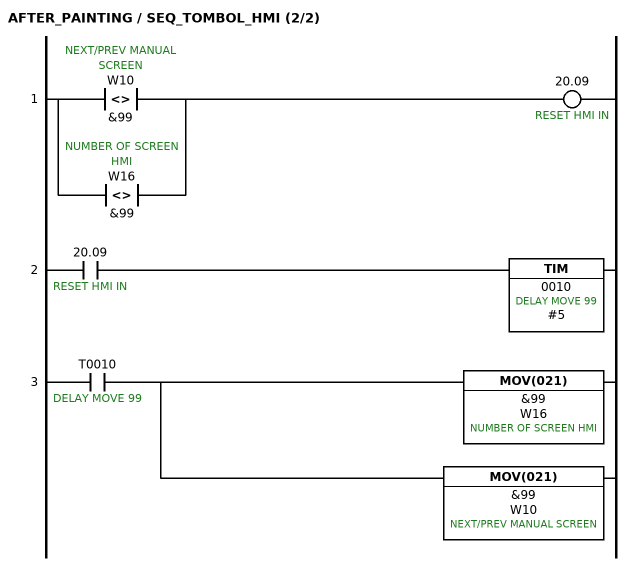
; [picture p48: AFTER_PAINTING / SEQ_TOMBOL_HMI, rungs 1-3]
; rung 1
LD<>(305) W10 &99  ; NEXT/PREV MANUAL SCREEN
OR<>(305) W16 &99  ; NUMBER OF SCREEN HMI
OUT 20.09  ; RESET HMI IN
; rung 2
LD 20.09  ; RESET HMI IN
TIM 0010 #5  ; DELAY MOVE 99
; rung 3
LD T0010  ; DELAY MOVE 99
MOV(021) &99 W16  ; NUMBER OF SCREEN HMI
MOV(021) &99 W10  ; NEXT/PREV MANUAL SCREEN

### Section AUTI

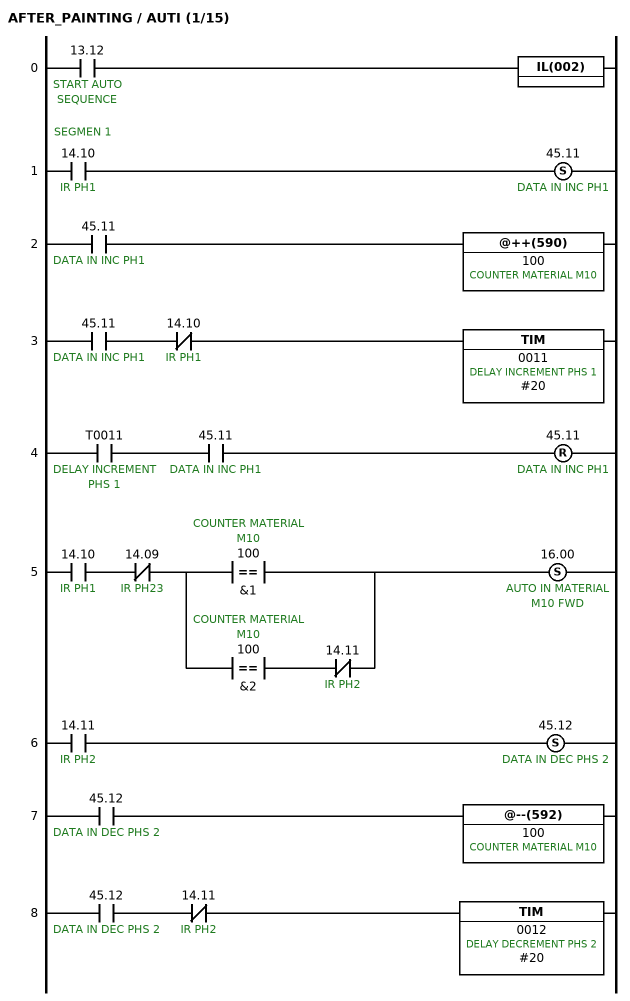
; rung 0
LD 13.12  ; START AUTO SEQUENCE
IL(002)
; rung 1: SEGMEN 1
LD 14.10  ; IR PH1
SET 45.11  ; DATA IN INC PH1
; rung 2
LD 45.11  ; DATA IN INC PH1
@++(590) 100  ; COUNTER MATERIAL M10
; rung 3
LD 45.11  ; DATA IN INC PH1
ANDNOT 14.10  ; IR PH1
TIM 0011 #20  ; DELAY INCREMENT PHS 1
; rung 4
LD T0011  ; DELAY INCREMENT PHS 1
AND 45.11  ; DATA IN INC PH1
RSET 45.11  ; DATA IN INC PH1
; rung 5
LD 14.10  ; IR PH1
ANDNOT 14.09  ; IR PH23
LD=(300) 100 &1  ; COUNTER MATERIAL M10
LD=(300) 100 &2  ; COUNTER MATERIAL M10
ANDNOT 14.11  ; IR PH2
ORLD
ANDLD
SET 16.00  ; AUTO IN MATERIAL M10 FWD
; rung 6
LD 14.11  ; IR PH2
SET 45.12  ; DATA IN DEC PHS 2
; rung 7
LD 45.12  ; DATA IN DEC PHS 2
@--(592) 100  ; COUNTER MATERIAL M10
; rung 8
LD 45.12  ; DATA IN DEC PHS 2
ANDNOT 14.11  ; IR PH2
TIM 0012 #20  ; DELAY DECREMENT PHS 2

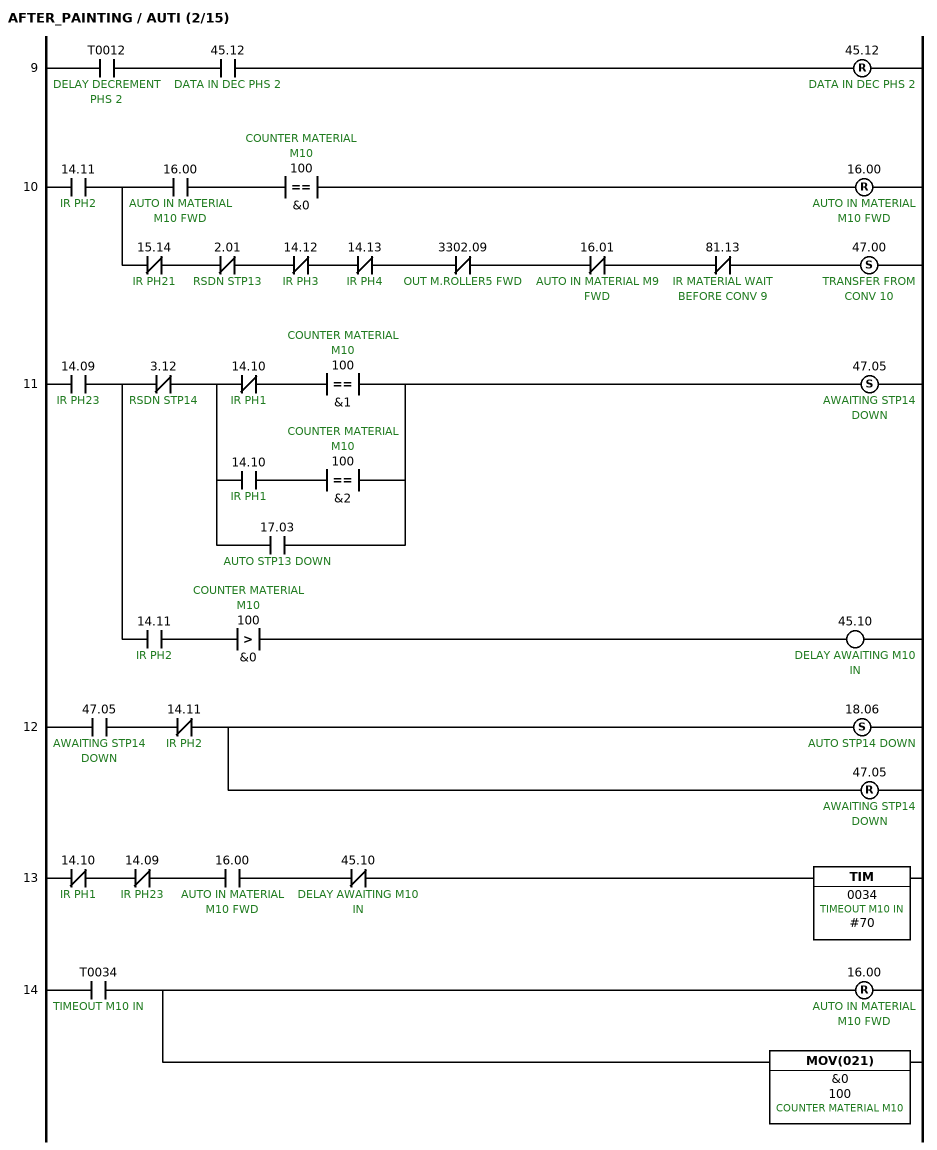
; rung 9
LD T0012  ; DELAY DECREMENT PHS 2
AND 45.12  ; DATA IN DEC PHS 2
RSET 45.12  ; DATA IN DEC PHS 2
; rung 10
LD 14.11  ; IR PH2
OUT TR0
AND 16.00  ; AUTO IN MATERIAL M10 FWD
AND=(300) 100 &0  ; COUNTER MATERIAL M10
RSET 16.00  ; AUTO IN MATERIAL M10 FWD
LD TR0
ANDNOT 15.14  ; IR PH21
ANDNOT 2.01  ; RSDN STP13
ANDNOT 14.12  ; IR PH3
ANDNOT 14.13  ; IR PH4
ANDNOT 3302.09  ; OUT M.ROLLER5 FWD
ANDNOT 16.01  ; AUTO IN MATERIAL M9 FWD
ANDNOT 81.13  ; IR MATERIAL WAIT BEFORE CONV 9
SET 47.00  ; TRANSFER FROM CONV 10
; rung 11
LD 14.09  ; IR PH23
OUT TR0
ANDNOT 3.12  ; RSDN STP14
LDNOT 14.10  ; IR PH1
AND=(300) 100 &1  ; COUNTER MATERIAL M10
LD 14.10  ; IR PH1
AND=(300) 100 &2  ; COUNTER MATERIAL M10
ORLD
OR 17.03  ; AUTO STP13 DOWN
ANDLD
SET 47.05  ; AWAITING STP14 DOWN
LD TR0
AND 14.11  ; IR PH2
AND>(320) 100 &0  ; COUNTER MATERIAL M10
OUT 45.10  ; DELAY AWAITING M10 IN
; rung 12
LD 47.05  ; AWAITING STP14 DOWN
ANDNOT 14.11  ; IR PH2
SET 18.06  ; AUTO STP14 DOWN
RSET 47.05  ; AWAITING STP14 DOWN
; rung 13
LDNOT 14.10  ; IR PH1
ANDNOT 14.09  ; IR PH23
AND 16.00  ; AUTO IN MATERIAL M10 FWD
ANDNOT 45.10  ; DELAY AWAITING M10 IN
TIM 0034 #70  ; TIMEOUT M10 IN
; rung 14
LD T0034  ; TIMEOUT M10 IN
RSET 16.00  ; AUTO IN MATERIAL M10 FWD
MOV(021) &0 100  ; COUNTER MATERIAL M10

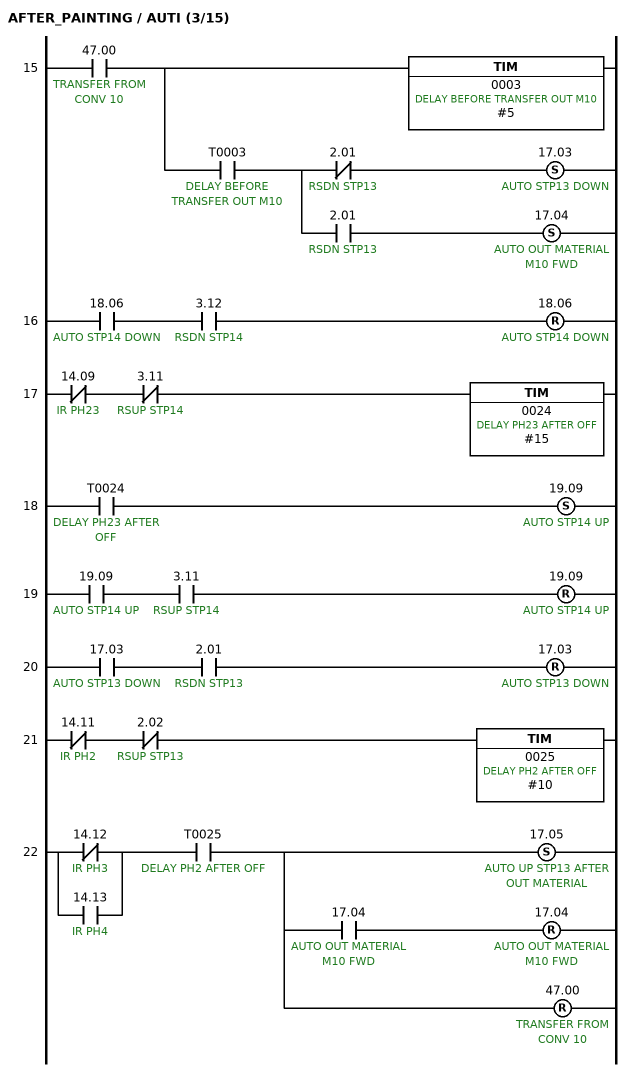
; rung 15
LD 47.00  ; TRANSFER FROM CONV 10
TIM 0003 #5  ; DELAY BEFORE TRANSFER OUT M10
AND T0003  ; DELAY BEFORE TRANSFER OUT M10
OUT TR0
ANDNOT 2.01  ; RSDN STP13
SET 17.03  ; AUTO STP13 DOWN
LD TR0
AND 2.01  ; RSDN STP13
SET 17.04  ; AUTO OUT MATERIAL M10 FWD
; rung 16
LD 18.06  ; AUTO STP14 DOWN
AND 3.12  ; RSDN STP14
RSET 18.06  ; AUTO STP14 DOWN
; rung 17
LDNOT 14.09  ; IR PH23
ANDNOT 3.11  ; RSUP STP14
TIM 0024 #15  ; DELAY PH23 AFTER OFF
; rung 18
LD T0024  ; DELAY PH23 AFTER OFF
SET 19.09  ; AUTO STP14 UP
; rung 19
LD 19.09  ; AUTO STP14 UP
AND 3.11  ; RSUP STP14
RSET 19.09  ; AUTO STP14 UP
; rung 20
LD 17.03  ; AUTO STP13 DOWN
AND 2.01  ; RSDN STP13
RSET 17.03  ; AUTO STP13 DOWN
; rung 21
LDNOT 14.11  ; IR PH2
ANDNOT 2.02  ; RSUP STP13
TIM 0025 #10  ; DELAY PH2 AFTER OFF
; rung 22
LDNOT 14.12  ; IR PH3
OR 14.13  ; IR PH4
AND T0025  ; DELAY PH2 AFTER OFF
OUT TR0
SET 17.05  ; AUTO UP STP13 AFTER OUT MATERIAL
AND 17.04  ; AUTO OUT MATERIAL M10 FWD
RSET 17.04  ; AUTO OUT MATERIAL M10 FWD
LD TR0
RSET 47.00  ; TRANSFER FROM CONV 10

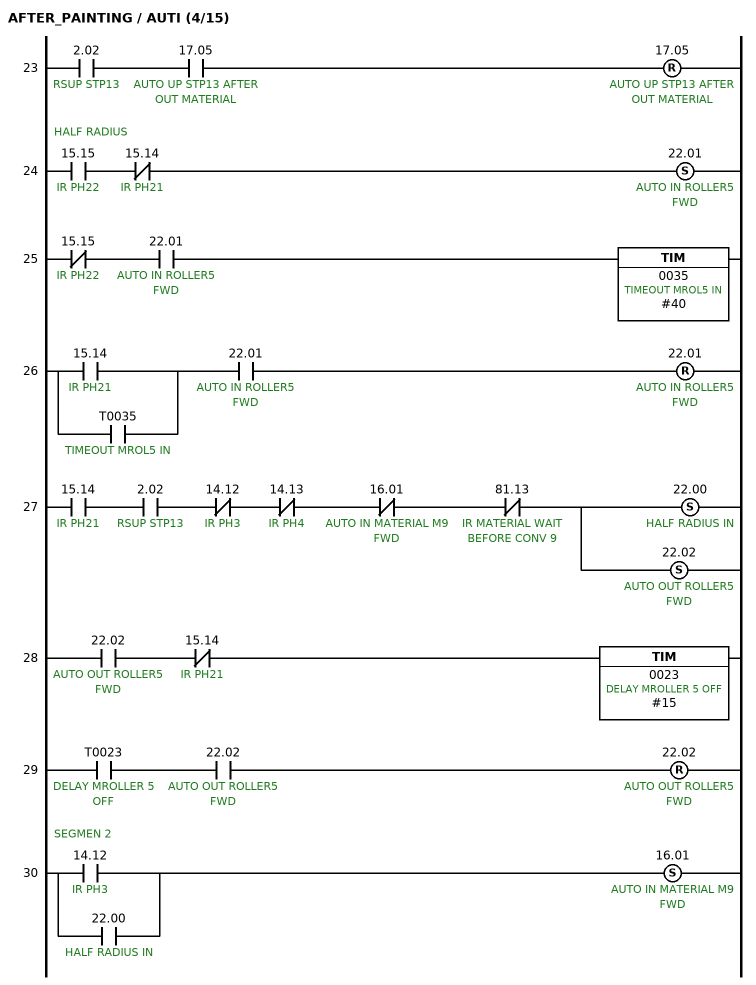
; rung 23
LD 2.02  ; RSUP STP13
AND 17.05  ; AUTO UP STP13 AFTER OUT MATERIAL
RSET 17.05  ; AUTO UP STP13 AFTER OUT MATERIAL
; rung 24: HALF RADIUS
LD 15.15  ; IR PH22
ANDNOT 15.14  ; IR PH21
SET 22.01  ; AUTO IN ROLLER5 FWD
; rung 25
LDNOT 15.15  ; IR PH22
AND 22.01  ; AUTO IN ROLLER5 FWD
TIM 0035 #40  ; TIMEOUT MROL5 IN
; rung 26
LD 15.14  ; IR PH21
OR T0035  ; TIMEOUT MROL5 IN
AND 22.01  ; AUTO IN ROLLER5 FWD
RSET 22.01  ; AUTO IN ROLLER5 FWD
; rung 27
LD 15.14  ; IR PH21
AND 2.02  ; RSUP STP13
ANDNOT 14.12  ; IR PH3
ANDNOT 14.13  ; IR PH4
ANDNOT 16.01  ; AUTO IN MATERIAL M9 FWD
ANDNOT 81.13  ; IR MATERIAL WAIT BEFORE CONV 9
SET 22.00  ; HALF RADIUS IN
SET 22.02  ; AUTO OUT ROLLER5 FWD
; rung 28
LD 22.02  ; AUTO OUT ROLLER5 FWD
ANDNOT 15.14  ; IR PH21
TIM 0023 #15  ; DELAY MROLLER 5 OFF
; rung 29
LD T0023  ; DELAY MROLLER 5 OFF
AND 22.02  ; AUTO OUT ROLLER5 FWD
RSET 22.02  ; AUTO OUT ROLLER5 FWD
; rung 30: SEGMEN 2
LD 14.12  ; IR PH3
OR 22.00  ; HALF RADIUS IN
SET 16.01  ; AUTO IN MATERIAL M9 FWD

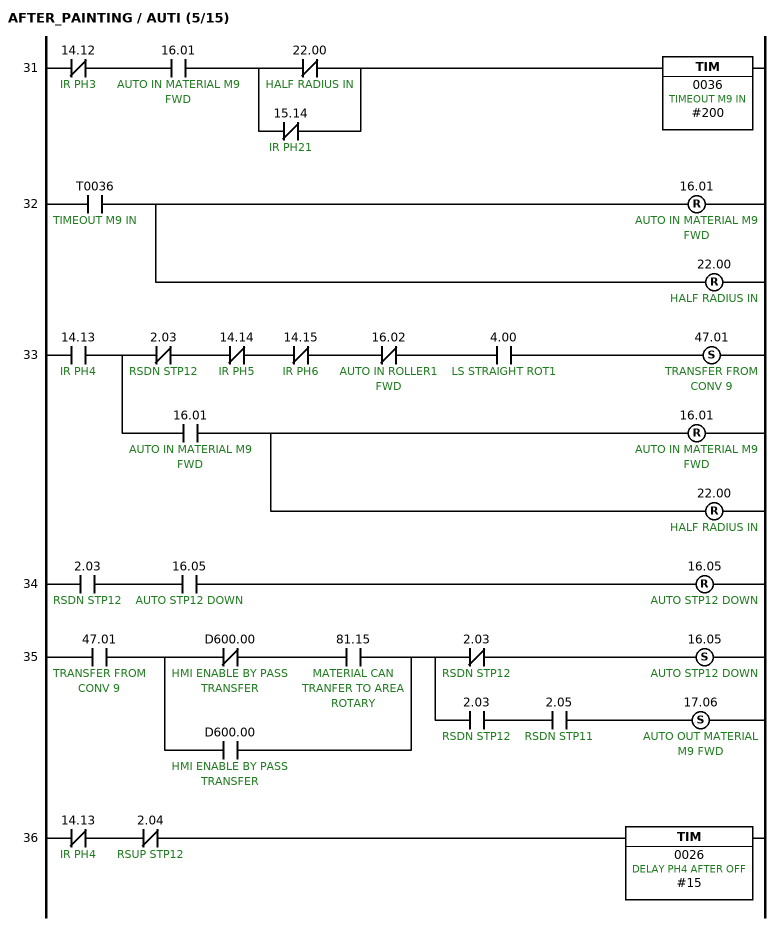
; rung 31
LDNOT 14.12  ; IR PH3
AND 16.01  ; AUTO IN MATERIAL M9 FWD
LDNOT 22.00  ; HALF RADIUS IN
ORNOT 15.14  ; IR PH21
ANDLD
TIM 0036 #200  ; TIMEOUT M9 IN
; rung 32
LD T0036  ; TIMEOUT M9 IN
RSET 16.01  ; AUTO IN MATERIAL M9 FWD
RSET 22.00  ; HALF RADIUS IN
; rung 33
LD 14.13  ; IR PH4
OUT TR0
ANDNOT 2.03  ; RSDN STP12
ANDNOT 14.14  ; IR PH5
ANDNOT 14.15  ; IR PH6
ANDNOT 16.02  ; AUTO IN ROLLER1 FWD
AND 4.00  ; LS STRAIGHT ROT1
SET 47.01  ; TRANSFER FROM CONV 9
LD TR0
AND 16.01  ; AUTO IN MATERIAL M9 FWD
RSET 16.01  ; AUTO IN MATERIAL M9 FWD
RSET 22.00  ; HALF RADIUS IN
; rung 34
LD 2.03  ; RSDN STP12
AND 16.05  ; AUTO STP12 DOWN
RSET 16.05  ; AUTO STP12 DOWN
; rung 35
LD 47.01  ; TRANSFER FROM CONV 9
LDNOT D600.00  ; HMI ENABLE BY PASS TRANSFER
AND 81.15  ; MATERIAL CAN TRANFER TO AREA ROTARY
OR D600.00  ; HMI ENABLE BY PASS TRANSFER
ANDLD
OUT TR0
ANDNOT 2.03  ; RSDN STP12
SET 16.05  ; AUTO STP12 DOWN
LD TR0
AND 2.03  ; RSDN STP12
AND 2.05  ; RSDN STP11
SET 17.06  ; AUTO OUT MATERIAL M9 FWD
; rung 36
LDNOT 14.13  ; IR PH4
ANDNOT 2.04  ; RSUP STP12
TIM 0026 #15  ; DELAY PH4 AFTER OFF

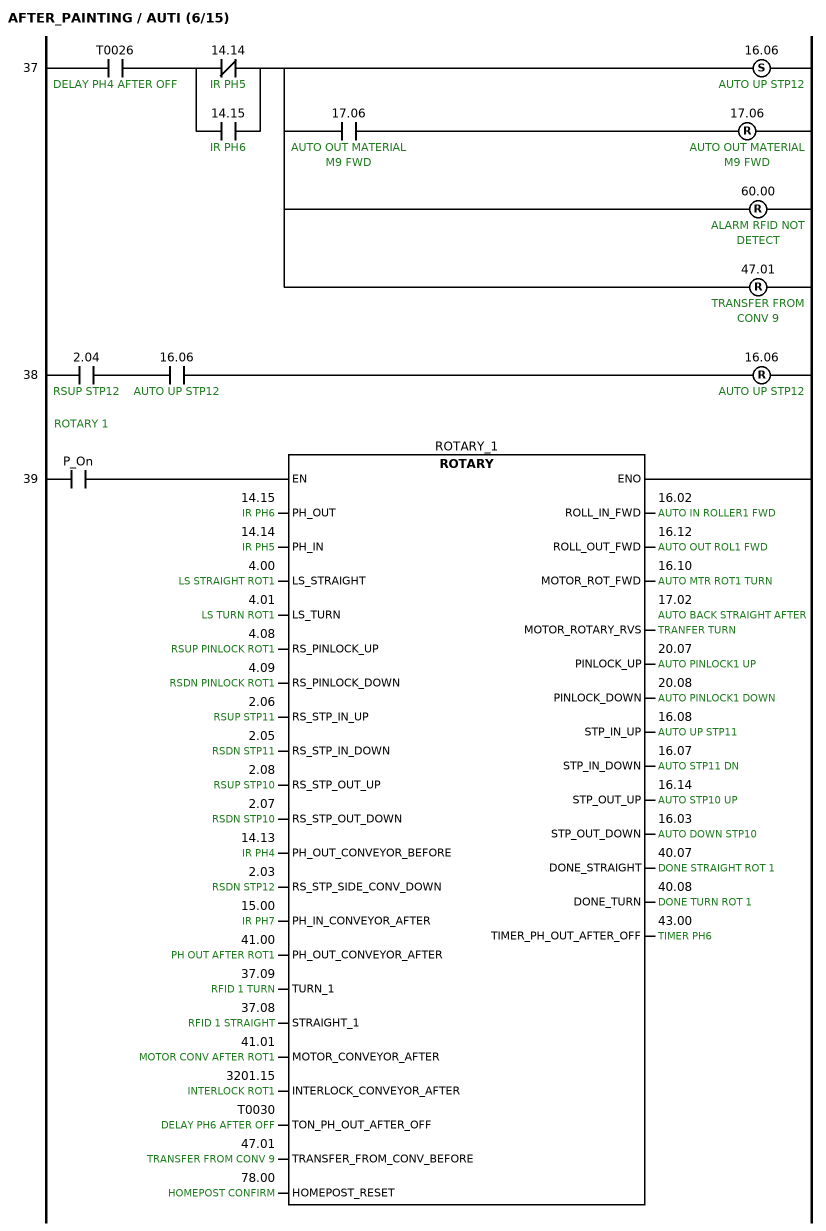
; rung 37
LD T0026  ; DELAY PH4 AFTER OFF
LDNOT 14.14  ; IR PH5
OR 14.15  ; IR PH6
ANDLD
OUT TR0
SET 16.06  ; AUTO UP STP12
AND 17.06  ; AUTO OUT MATERIAL M9 FWD
RSET 17.06  ; AUTO OUT MATERIAL M9 FWD
LD TR0
RSET 60.00  ; ALARM RFID NOT DETECT
RSET 47.01  ; TRANSFER FROM CONV 9
; rung 38
LD 2.04  ; RSUP STP12
AND 16.06  ; AUTO UP STP12
RSET 16.06  ; AUTO UP STP12
; rung 39: ROTARY 1
LD P_On
CALL ROTARY_1 : ROTARY (PH_OUT := 14.15, PH_IN := 14.14, LS_STRAIGHT := 4.00, LS_TURN := 4.01, RS_PINLOCK_UP := 4.08, RS_PINLOCK_DOWN := 4.09, RS_STP_IN_UP := 2.06, RS_STP_IN_DOWN := 2.05, RS_STP_OUT_UP := 2.08, RS_STP_OUT_DOWN := 2.07, PH_OUT_CONVEYOR_BEFORE := 14.13, RS_STP_SIDE_CONV_DOWN := 2.03, PH_IN_CONVEYOR_AFTER := 15.00, PH_OUT_CONVEYOR_AFTER := 41.00, TURN_1 := 37.09, STRAIGHT_1 := 37.08, MOTOR_CONVEYOR_AFTER := 41.01, INTERLOCK_CONVEYOR_AFTER := 3201.15, TON_PH_OUT_AFTER_OFF := T0030, TRANSFER_FROM_CONV_BEFORE := 47.01, HOMEPOST_RESET := 78.00, ROLL_IN_FWD => 16.02, ROLL_OUT_FWD => 16.12, MOTOR_ROT_FWD => 16.10, MOTOR_ROTARY_RVS => 17.02, PINLOCK_UP => 20.07, PINLOCK_DOWN => 20.08, STP_IN_UP => 16.08, STP_IN_DOWN => 16.07, STP_OUT_UP => 16.14, STP_OUT_DOWN => 16.03, DONE_STRAIGHT => 40.07, DONE_TURN => 40.08, TIMER_PH_OUT_AFTER_OFF => 43.00)  ; IR PH6, IR PH5, LS STRAIGHT ROT1, LS TURN ROT1, RSUP PINLOCK ROT1, RSDN PINLOCK ROT1, RSUP STP11, RSDN STP11, RSUP STP10, RSDN STP10, IR PH4, RSDN STP12, IR PH7, PH OUT AFTER ROT1, RFID 1 TURN, RFID 1 STRAIGHT, MOTOR CONV AFTER ROT1, INTERLOCK ROT1, DELAY PH6 AFTER OFF, TRANSFER FROM CONV 9, HOMEPOST CONFIRM, AUTO IN ROLLER1 FWD, AUTO OUT ROL1 FWD, AUTO MTR ROT1 TURN, AUTO BACK STRAIGHT AFTER TRANFER TURN, AUTO PINLOCK1 UP, AUTO PINLOCK1 DOWN, AUTO UP STP11, AUTO STP11 DN, AUTO STP10 UP, AUTO DOWN STP10, DONE STRAIGHT ROT 1, DONE TURN ROT 1, TIMER PH6

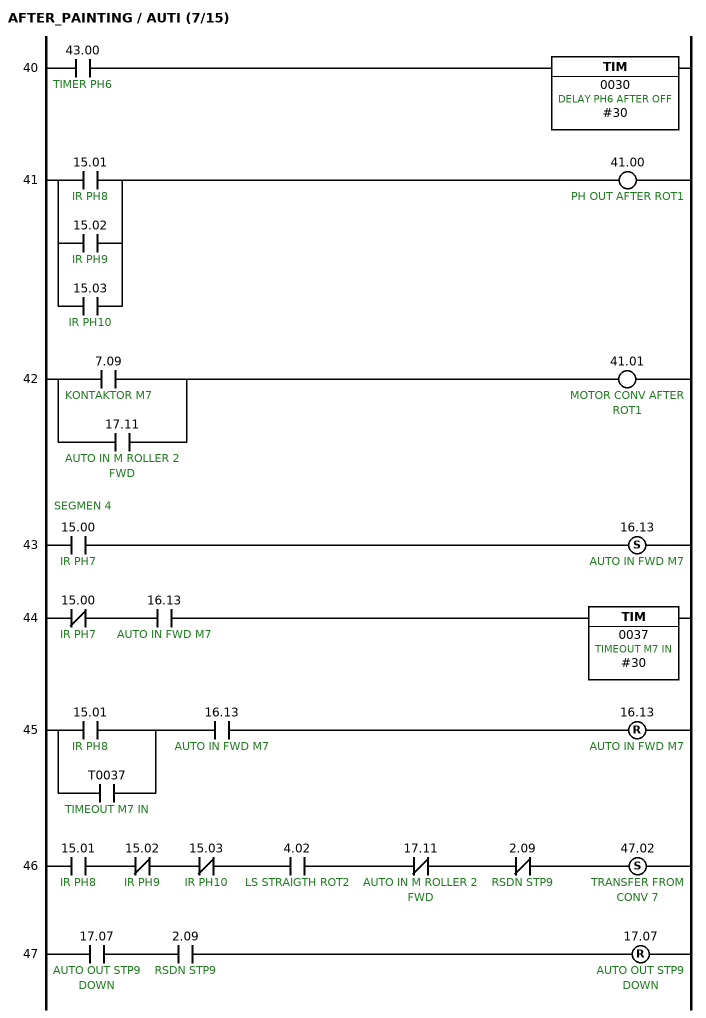
; rung 40
LD 43.00  ; TIMER PH6
TIM 0030 #30  ; DELAY PH6 AFTER OFF
; rung 41
LD 15.01  ; IR PH8
OR 15.02  ; IR PH9
OR 15.03  ; IR PH10
OUT 41.00  ; PH OUT AFTER ROT1
; rung 42
LD 7.09  ; KONTAKTOR M7
OR 17.11  ; AUTO IN M ROLLER 2 FWD
OUT 41.01  ; MOTOR CONV AFTER ROT1
; rung 43: SEGMEN 4
LD 15.00  ; IR PH7
SET 16.13  ; AUTO IN FWD M7
; rung 44
LDNOT 15.00  ; IR PH7
AND 16.13  ; AUTO IN FWD M7
TIM 0037 #30  ; TIMEOUT M7 IN
; rung 45
LD 15.01  ; IR PH8
OR T0037  ; TIMEOUT M7 IN
AND 16.13  ; AUTO IN FWD M7
RSET 16.13  ; AUTO IN FWD M7
; rung 46
LD 15.01  ; IR PH8
ANDNOT 15.02  ; IR PH9
ANDNOT 15.03  ; IR PH10
AND 4.02  ; LS STRAIGTH ROT2
ANDNOT 17.11  ; AUTO IN M ROLLER 2 FWD
ANDNOT 2.09  ; RSDN STP9
SET 47.02  ; TRANSFER FROM CONV 7
; rung 47
LD 17.07  ; AUTO OUT STP9 DOWN
AND 2.09  ; RSDN STP9
RSET 17.07  ; AUTO OUT STP9 DOWN

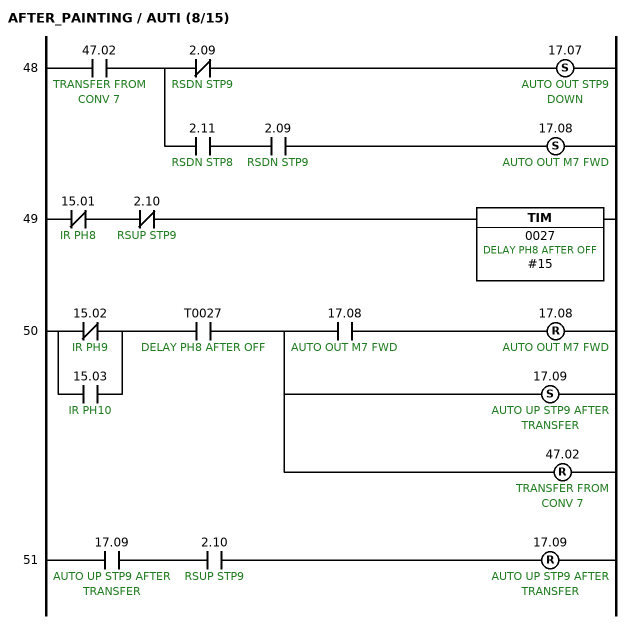
; rung 48
LD 47.02  ; TRANSFER FROM CONV 7
OUT TR0
ANDNOT 2.09  ; RSDN STP9
SET 17.07  ; AUTO OUT STP9 DOWN
LD TR0
AND 2.11  ; RSDN STP8
AND 2.09  ; RSDN STP9
SET 17.08  ; AUTO OUT M7 FWD
; rung 49
LDNOT 15.01  ; IR PH8
ANDNOT 2.10  ; RSUP STP9
TIM 0027 #15  ; DELAY PH8 AFTER OFF
; rung 50
LDNOT 15.02  ; IR PH9
OR 15.03  ; IR PH10
AND T0027  ; DELAY PH8 AFTER OFF
OUT TR0
AND 17.08  ; AUTO OUT M7 FWD
RSET 17.08  ; AUTO OUT M7 FWD
LD TR0
SET 17.09  ; AUTO UP STP9 AFTER TRANSFER
RSET 47.02  ; TRANSFER FROM CONV 7
; rung 51
LD 17.09  ; AUTO UP STP9 AFTER TRANSFER
AND 2.10  ; RSUP STP9
RSET 17.09  ; AUTO UP STP9 AFTER TRANSFER

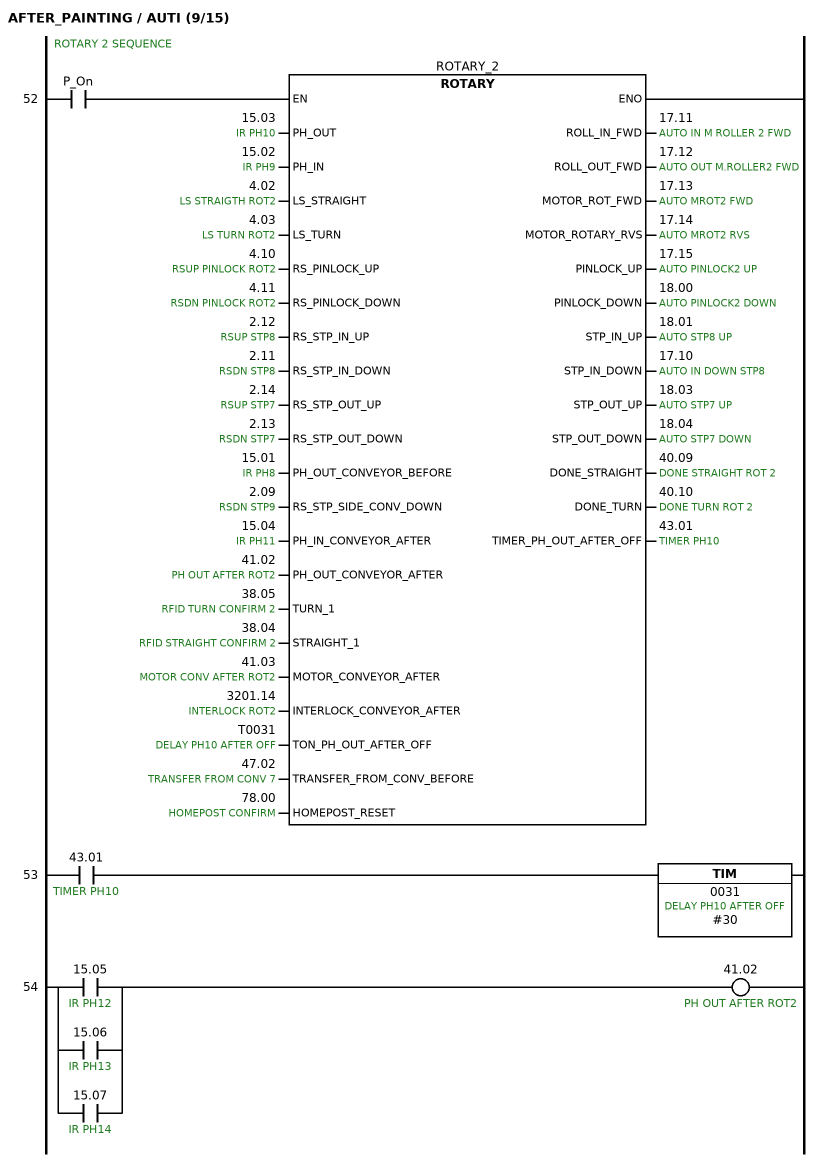
; rung 52: ROTARY 2 SEQUENCE
LD P_On
CALL ROTARY_2 : ROTARY (PH_OUT := 15.03, PH_IN := 15.02, LS_STRAIGHT := 4.02, LS_TURN := 4.03, RS_PINLOCK_UP := 4.10, RS_PINLOCK_DOWN := 4.11, RS_STP_IN_UP := 2.12, RS_STP_IN_DOWN := 2.11, RS_STP_OUT_UP := 2.14, RS_STP_OUT_DOWN := 2.13, PH_OUT_CONVEYOR_BEFORE := 15.01, RS_STP_SIDE_CONV_DOWN := 2.09, PH_IN_CONVEYOR_AFTER := 15.04, PH_OUT_CONVEYOR_AFTER := 41.02, TURN_1 := 38.05, STRAIGHT_1 := 38.04, MOTOR_CONVEYOR_AFTER := 41.03, INTERLOCK_CONVEYOR_AFTER := 3201.14, TON_PH_OUT_AFTER_OFF := T0031, TRANSFER_FROM_CONV_BEFORE := 47.02, HOMEPOST_RESET := 78.00, ROLL_IN_FWD => 17.11, ROLL_OUT_FWD => 17.12, MOTOR_ROT_FWD => 17.13, MOTOR_ROTARY_RVS => 17.14, PINLOCK_UP => 17.15, PINLOCK_DOWN => 18.00, STP_IN_UP => 18.01, STP_IN_DOWN => 17.10, STP_OUT_UP => 18.03, STP_OUT_DOWN => 18.04, DONE_STRAIGHT => 40.09, DONE_TURN => 40.10, TIMER_PH_OUT_AFTER_OFF => 43.01)  ; IR PH10, IR PH9, LS STRAIGTH ROT2, LS TURN ROT2, RSUP PINLOCK ROT2, RSDN PINLOCK ROT2, RSUP STP8, RSDN STP8, RSUP STP7, RSDN STP7, IR PH8, RSDN STP9, IR PH11, PH OUT AFTER ROT2, RFID TURN CONFIRM 2, RFID STRAIGHT CONFIRM 2, MOTOR CONV AFTER ROT2, INTERLOCK ROT2, DELAY PH10 AFTER OFF, TRANSFER FROM CONV 7, HOMEPOST CONFIRM, AUTO IN M ROLLER 2 FWD, AUTO OUT M.ROLLER2 FWD, AUTO MROT2 FWD, AUTO MROT2 RVS, AUTO PINLOCK2 UP, AUTO PINLOCK2 DOWN, AUTO STP8 UP, AUTO IN DOWN STP8, AUTO STP7 UP, AUTO STP7 DOWN, DONE STRAIGHT ROT 2, DONE TURN ROT 2, TIMER PH10
; rung 53
LD 43.01  ; TIMER PH10
TIM 0031 #30  ; DELAY PH10 AFTER OFF
; rung 54
LD 15.05  ; IR PH12
OR 15.06  ; IR PH13
OR 15.07  ; IR PH14
OUT 41.02  ; PH OUT AFTER ROT2

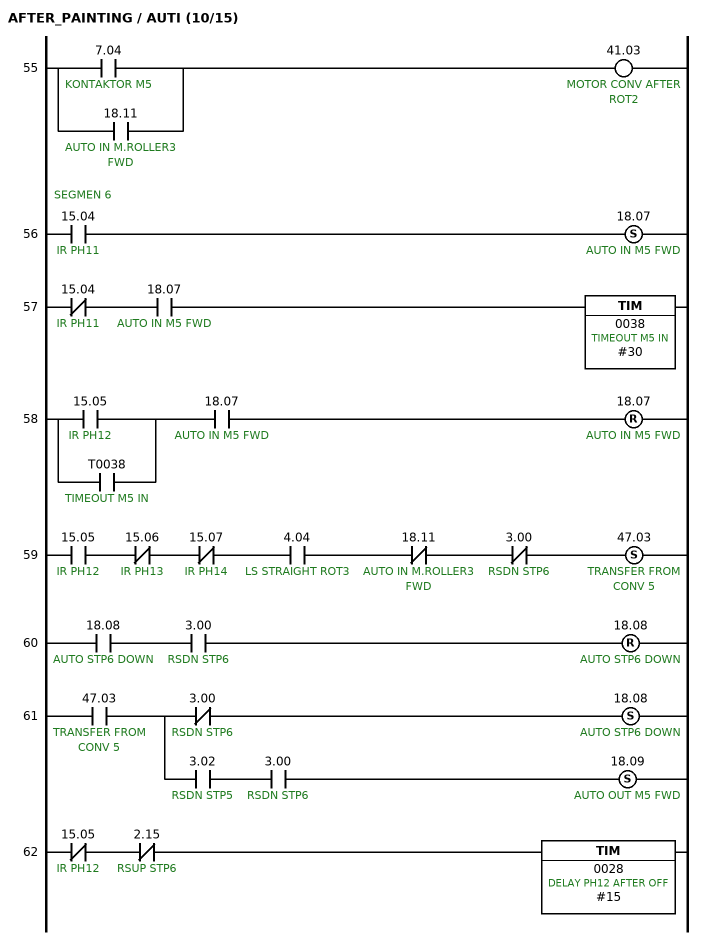
; rung 55
LD 7.04  ; KONTAKTOR M5
OR 18.11  ; AUTO IN M.ROLLER3 FWD
OUT 41.03  ; MOTOR CONV AFTER ROT2
; rung 56: SEGMEN 6
LD 15.04  ; IR PH11
SET 18.07  ; AUTO IN M5 FWD
; rung 57
LDNOT 15.04  ; IR PH11
AND 18.07  ; AUTO IN M5 FWD
TIM 0038 #30  ; TIMEOUT M5 IN
; rung 58
LD 15.05  ; IR PH12
OR T0038  ; TIMEOUT M5 IN
AND 18.07  ; AUTO IN M5 FWD
RSET 18.07  ; AUTO IN M5 FWD
; rung 59
LD 15.05  ; IR PH12
ANDNOT 15.06  ; IR PH13
ANDNOT 15.07  ; IR PH14
AND 4.04  ; LS STRAIGHT ROT3
ANDNOT 18.11  ; AUTO IN M.ROLLER3 FWD
ANDNOT 3.00  ; RSDN STP6
SET 47.03  ; TRANSFER FROM CONV 5
; rung 60
LD 18.08  ; AUTO STP6 DOWN
AND 3.00  ; RSDN STP6
RSET 18.08  ; AUTO STP6 DOWN
; rung 61
LD 47.03  ; TRANSFER FROM CONV 5
OUT TR0
ANDNOT 3.00  ; RSDN STP6
SET 18.08  ; AUTO STP6 DOWN
LD TR0
AND 3.02  ; RSDN STP5
AND 3.00  ; RSDN STP6
SET 18.09  ; AUTO OUT M5 FWD
; rung 62
LDNOT 15.05  ; IR PH12
ANDNOT 2.15  ; RSUP STP6
TIM 0028 #15  ; DELAY PH12 AFTER OFF

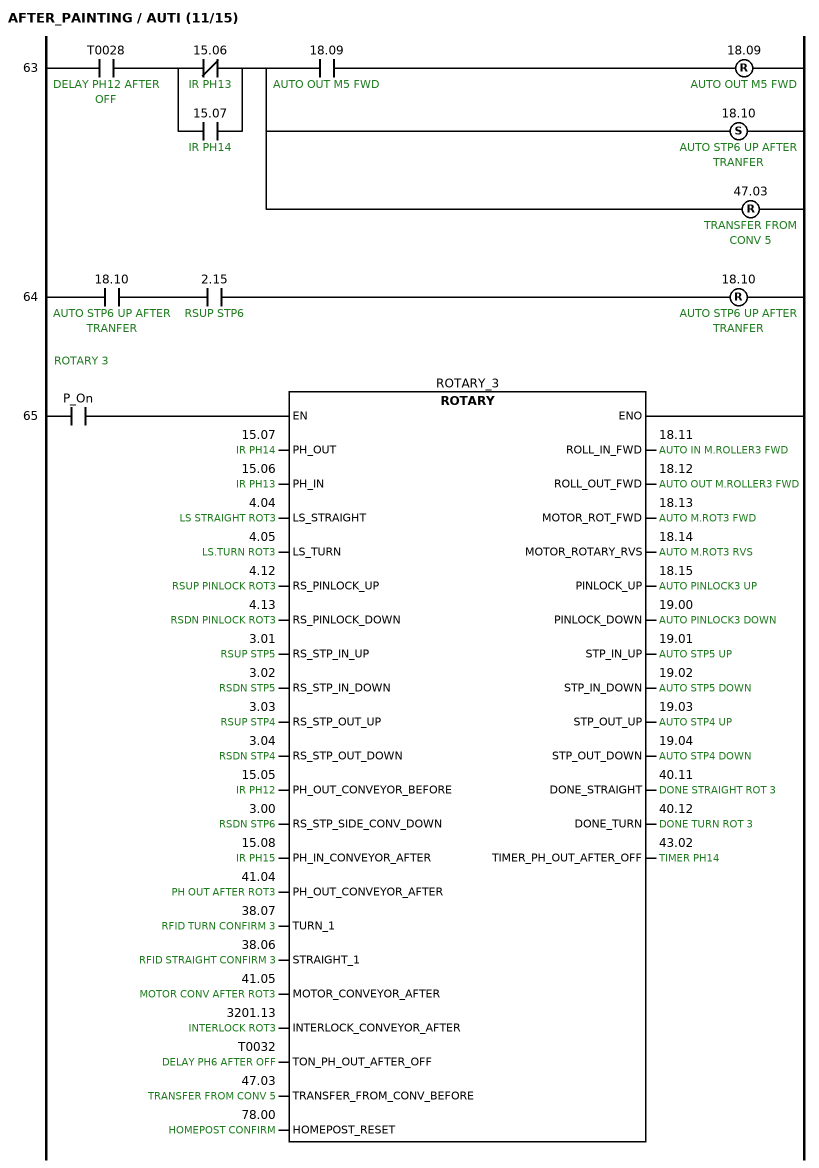
; rung 63
LD T0028  ; DELAY PH12 AFTER OFF
LDNOT 15.06  ; IR PH13
OR 15.07  ; IR PH14
ANDLD
OUT TR0
AND 18.09  ; AUTO OUT M5 FWD
RSET 18.09  ; AUTO OUT M5 FWD
LD TR0
SET 18.10  ; AUTO STP6 UP AFTER TRANFER
RSET 47.03  ; TRANSFER FROM CONV 5
; rung 64
LD 18.10  ; AUTO STP6 UP AFTER TRANFER
AND 2.15  ; RSUP STP6
RSET 18.10  ; AUTO STP6 UP AFTER TRANFER
; rung 65: ROTARY 3
LD P_On
CALL ROTARY_3 : ROTARY (PH_OUT := 15.07, PH_IN := 15.06, LS_STRAIGHT := 4.04, LS_TURN := 4.05, RS_PINLOCK_UP := 4.12, RS_PINLOCK_DOWN := 4.13, RS_STP_IN_UP := 3.01, RS_STP_IN_DOWN := 3.02, RS_STP_OUT_UP := 3.03, RS_STP_OUT_DOWN := 3.04, PH_OUT_CONVEYOR_BEFORE := 15.05, RS_STP_SIDE_CONV_DOWN := 3.00, PH_IN_CONVEYOR_AFTER := 15.08, PH_OUT_CONVEYOR_AFTER := 41.04, TURN_1 := 38.07, STRAIGHT_1 := 38.06, MOTOR_CONVEYOR_AFTER := 41.05, INTERLOCK_CONVEYOR_AFTER := 3201.13, TON_PH_OUT_AFTER_OFF := T0032, TRANSFER_FROM_CONV_BEFORE := 47.03, HOMEPOST_RESET := 78.00, ROLL_IN_FWD => 18.11, ROLL_OUT_FWD => 18.12, MOTOR_ROT_FWD => 18.13, MOTOR_ROTARY_RVS => 18.14, PINLOCK_UP => 18.15, PINLOCK_DOWN => 19.00, STP_IN_UP => 19.01, STP_IN_DOWN => 19.02, STP_OUT_UP => 19.03, STP_OUT_DOWN => 19.04, DONE_STRAIGHT => 40.11, DONE_TURN => 40.12, TIMER_PH_OUT_AFTER_OFF => 43.02)  ; IR PH14, IR PH13, LS STRAIGHT ROT3, LS.TURN ROT3, RSUP PINLOCK ROT3, RSDN PINLOCK ROT3, RSUP STP5, RSDN STP5, RSUP STP4, RSDN STP4, IR PH12, RSDN STP6, IR PH15, PH OUT AFTER ROT3, RFID TURN CONFIRM 3, RFID STRAIGHT CONFIRM 3, MOTOR CONV AFTER ROT3, INTERLOCK ROT3, DELAY PH6 AFTER OFF, TRANSFER FROM CONV 5, HOMEPOST CONFIRM, AUTO IN M.ROLLER3 FWD, AUTO OUT M.ROLLER3 FWD, AUTO M.ROT3 FWD, AUTO M.ROT3 RVS, AUTO PINLOCK3 UP, AUTO PINLOCK3 DOWN, AUTO STP5 UP, AUTO STP5 DOWN, AUTO STP4 UP, AUTO STP4 DOWN, DONE STRAIGHT ROT 3, DONE TURN ROT 3, TIMER PH14

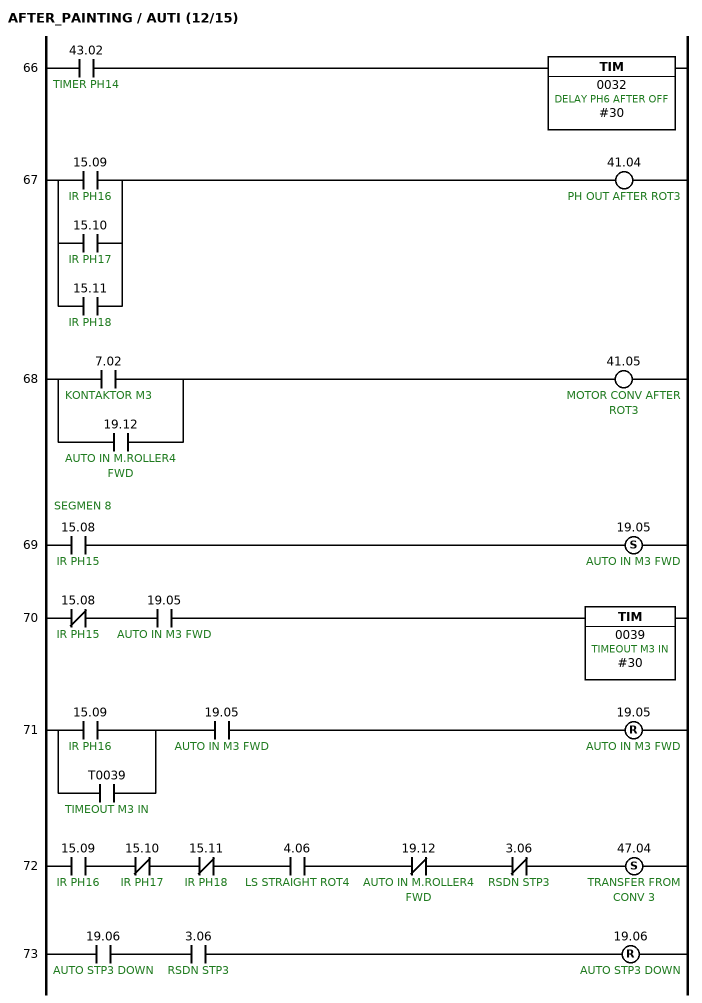
; rung 66
LD 43.02  ; TIMER PH14
TIM 0032 #30  ; DELAY PH6 AFTER OFF
; rung 67
LD 15.09  ; IR PH16
OR 15.10  ; IR PH17
OR 15.11  ; IR PH18
OUT 41.04  ; PH OUT AFTER ROT3
; rung 68
LD 7.02  ; KONTAKTOR M3
OR 19.12  ; AUTO IN M.ROLLER4 FWD
OUT 41.05  ; MOTOR CONV AFTER ROT3
; rung 69: SEGMEN 8
LD 15.08  ; IR PH15
SET 19.05  ; AUTO IN M3 FWD
; rung 70
LDNOT 15.08  ; IR PH15
AND 19.05  ; AUTO IN M3 FWD
TIM 0039 #30  ; TIMEOUT M3 IN
; rung 71
LD 15.09  ; IR PH16
OR T0039  ; TIMEOUT M3 IN
AND 19.05  ; AUTO IN M3 FWD
RSET 19.05  ; AUTO IN M3 FWD
; rung 72
LD 15.09  ; IR PH16
ANDNOT 15.10  ; IR PH17
ANDNOT 15.11  ; IR PH18
AND 4.06  ; LS STRAIGHT ROT4
ANDNOT 19.12  ; AUTO IN M.ROLLER4 FWD
ANDNOT 3.06  ; RSDN STP3
SET 47.04  ; TRANSFER FROM CONV 3
; rung 73
LD 19.06  ; AUTO STP3 DOWN
AND 3.06  ; RSDN STP3
RSET 19.06  ; AUTO STP3 DOWN

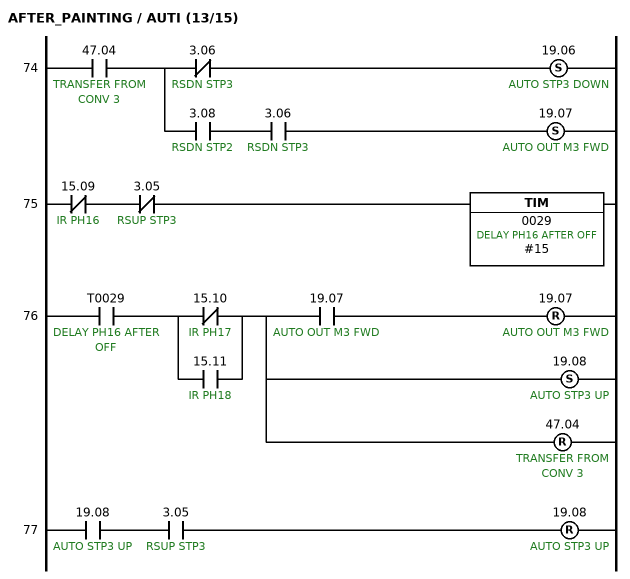
; rung 74
LD 47.04  ; TRANSFER FROM CONV 3
OUT TR0
ANDNOT 3.06  ; RSDN STP3
SET 19.06  ; AUTO STP3 DOWN
LD TR0
AND 3.08  ; RSDN STP2
AND 3.06  ; RSDN STP3
SET 19.07  ; AUTO OUT M3 FWD
; rung 75
LDNOT 15.09  ; IR PH16
ANDNOT 3.05  ; RSUP STP3
TIM 0029 #15  ; DELAY PH16 AFTER OFF
; rung 76
LD T0029  ; DELAY PH16 AFTER OFF
LDNOT 15.10  ; IR PH17
OR 15.11  ; IR PH18
ANDLD
OUT TR0
AND 19.07  ; AUTO OUT M3 FWD
RSET 19.07  ; AUTO OUT M3 FWD
LD TR0
SET 19.08  ; AUTO STP3 UP
RSET 47.04  ; TRANSFER FROM CONV 3
; rung 77
LD 19.08  ; AUTO STP3 UP
AND 3.05  ; RSUP STP3
RSET 19.08  ; AUTO STP3 UP

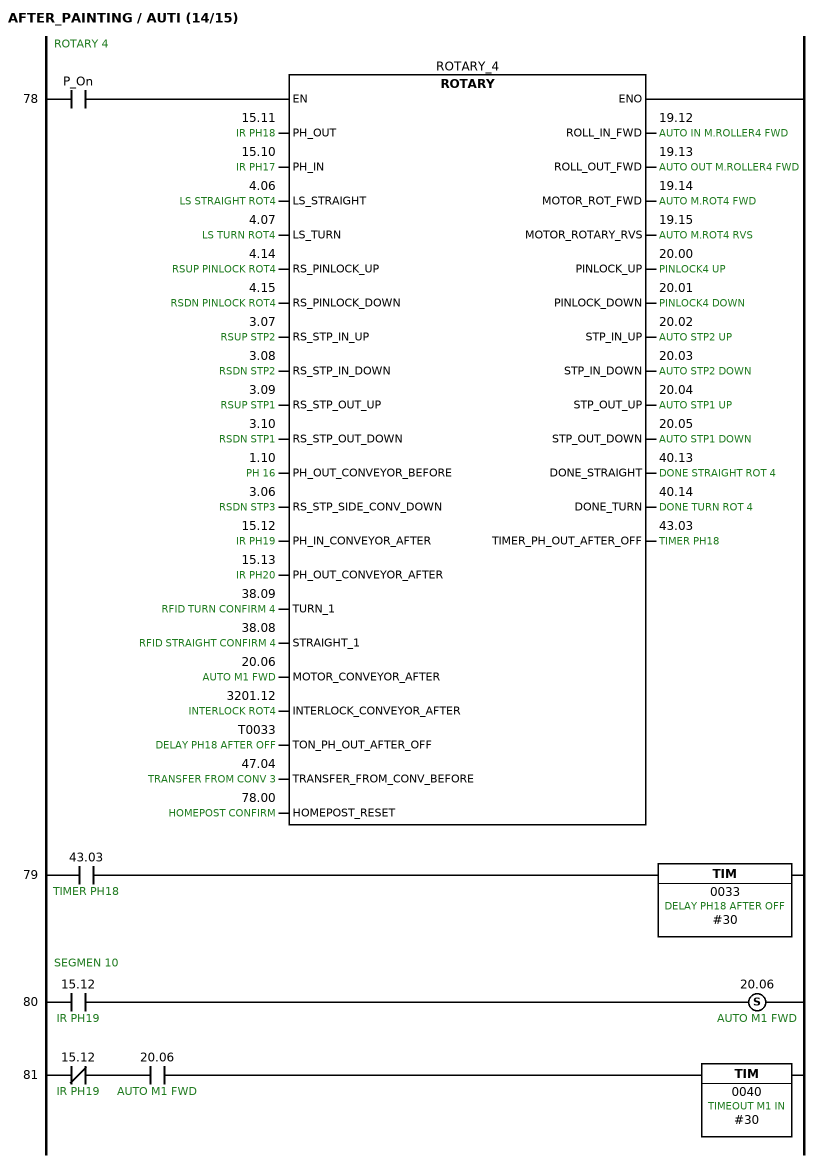
; rung 78: ROTARY 4
LD P_On
CALL ROTARY_4 : ROTARY (PH_OUT := 15.11, PH_IN := 15.10, LS_STRAIGHT := 4.06, LS_TURN := 4.07, RS_PINLOCK_UP := 4.14, RS_PINLOCK_DOWN := 4.15, RS_STP_IN_UP := 3.07, RS_STP_IN_DOWN := 3.08, RS_STP_OUT_UP := 3.09, RS_STP_OUT_DOWN := 3.10, PH_OUT_CONVEYOR_BEFORE := 1.10, RS_STP_SIDE_CONV_DOWN := 3.06, PH_IN_CONVEYOR_AFTER := 15.12, PH_OUT_CONVEYOR_AFTER := 15.13, TURN_1 := 38.09, STRAIGHT_1 := 38.08, MOTOR_CONVEYOR_AFTER := 20.06, INTERLOCK_CONVEYOR_AFTER := 3201.12, TON_PH_OUT_AFTER_OFF := T0033, TRANSFER_FROM_CONV_BEFORE := 47.04, HOMEPOST_RESET := 78.00, ROLL_IN_FWD => 19.12, ROLL_OUT_FWD => 19.13, MOTOR_ROT_FWD => 19.14, MOTOR_ROTARY_RVS => 19.15, PINLOCK_UP => 20.00, PINLOCK_DOWN => 20.01, STP_IN_UP => 20.02, STP_IN_DOWN => 20.03, STP_OUT_UP => 20.04, STP_OUT_DOWN => 20.05, DONE_STRAIGHT => 40.13, DONE_TURN => 40.14, TIMER_PH_OUT_AFTER_OFF => 43.03)  ; IR PH18, IR PH17, LS STRAIGHT ROT4, LS TURN ROT4, RSUP PINLOCK ROT4, RSDN PINLOCK ROT4, RSUP STP2, RSDN STP2, RSUP STP1, RSDN STP1, PH 16, RSDN STP3, IR PH19, IR PH20, RFID TURN CONFIRM 4, RFID STRAIGHT CONFIRM 4, AUTO M1 FWD, INTERLOCK ROT4, DELAY PH18 AFTER OFF, TRANSFER FROM CONV 3, HOMEPOST CONFIRM, AUTO IN M.ROLLER4 FWD, AUTO OUT M.ROLLER4 FWD, AUTO M.ROT4 FWD, AUTO M.ROT4 RVS, PINLOCK4 UP, PINLOCK4 DOWN, AUTO STP2 UP, AUTO STP2 DOWN, AUTO STP1 UP, AUTO STP1 DOWN, DONE STRAIGHT ROT 4, DONE TURN ROT 4, TIMER PH18
; rung 79
LD 43.03  ; TIMER PH18
TIM 0033 #30  ; DELAY PH18 AFTER OFF
; rung 80: SEGMEN 10
LD 15.12  ; IR PH19
SET 20.06  ; AUTO M1 FWD
; rung 81
LDNOT 15.12  ; IR PH19
AND 20.06  ; AUTO M1 FWD
TIM 0040 #30  ; TIMEOUT M1 IN

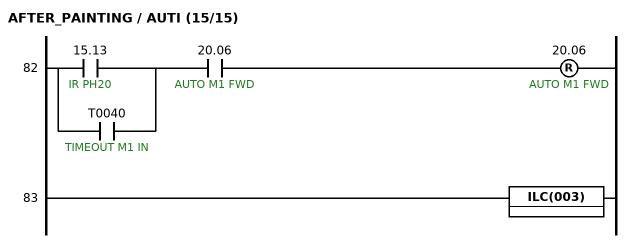
; rung 82
LD 15.13  ; IR PH20
OR T0040  ; TIMEOUT M1 IN
AND 20.06  ; AUTO M1 FWD
RSET 20.06  ; AUTO M1 FWD
; rung 83
ILC(003)

### Section SERIAL

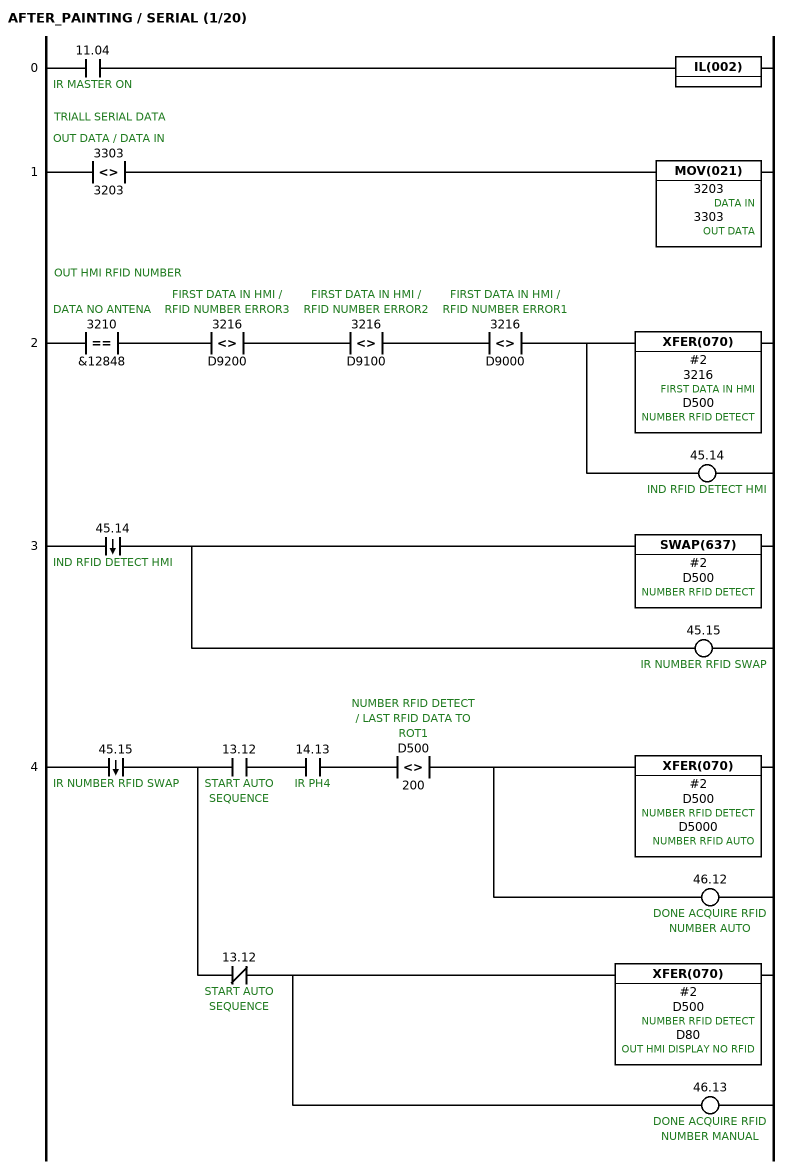
; rung 0
LD 11.04  ; IR MASTER ON
IL(002)
; rung 1: TRIALL SERIAL DATA
LD<>(305) 3303 3203  ; OUT DATA, DATA IN
MOV(021) 3203 3303  ; DATA IN, OUT DATA
; rung 2: OUT HMI RFID NUMBER
LD=(300) 3210 &12848  ; DATA NO ANTENA
AND<>(305) 3216 D9200  ; FIRST DATA IN HMI, RFID NUMBER ERROR3
AND<>(305) 3216 D9100  ; FIRST DATA IN HMI, RFID NUMBER ERROR2
AND<>(305) 3216 D9000  ; FIRST DATA IN HMI, RFID NUMBER ERROR1
XFER(070) #2 3216 D500  ; FIRST DATA IN HMI, NUMBER RFID DETECT
OUT 45.14  ; IND RFID DETECT HMI
; rung 3
%LD 45.14  ; IND RFID DETECT HMI
SWAP(637) #2 D500  ; NUMBER RFID DETECT
OUT 45.15  ; IR NUMBER RFID SWAP
; rung 4
%LD 45.15  ; IR NUMBER RFID SWAP
OUT TR0
AND 13.12  ; START AUTO SEQUENCE
AND 14.13  ; IR PH4
AND<>(305) D500 200  ; NUMBER RFID DETECT, LAST RFID DATA TO ROT1
XFER(070) #2 D500 D5000  ; NUMBER RFID DETECT, NUMBER RFID AUTO
OUT 46.12  ; DONE ACQUIRE RFID NUMBER AUTO
LD TR0
ANDNOT 13.12  ; START AUTO SEQUENCE
XFER(070) #2 D500 D80  ; NUMBER RFID DETECT, OUT HMI DISPLAY NO RFID
OUT 46.13  ; DONE ACQUIRE RFID NUMBER MANUAL

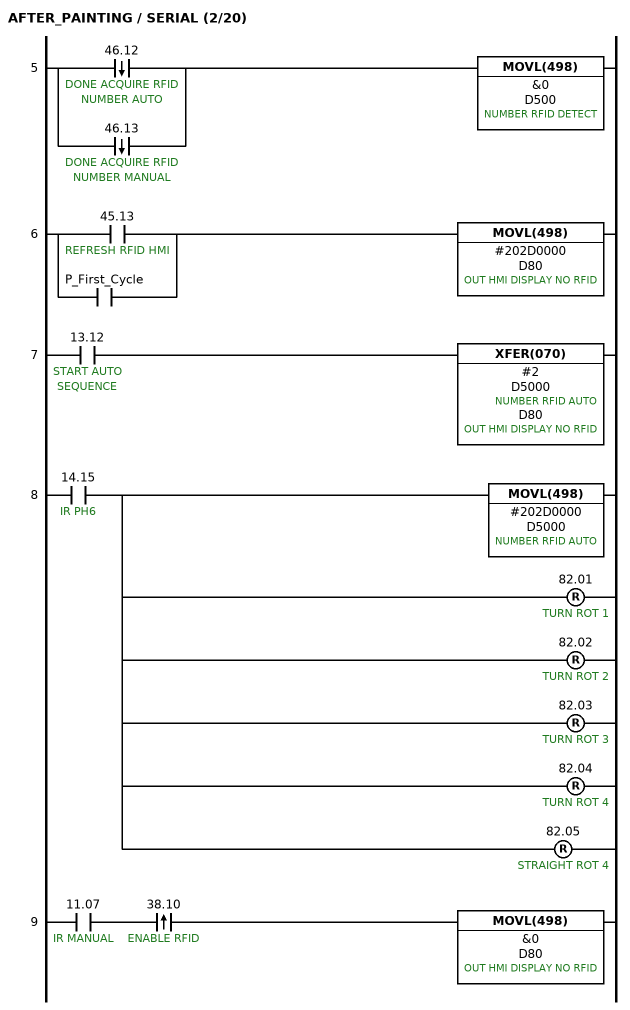
; rung 5
%LD 46.12  ; DONE ACQUIRE RFID NUMBER AUTO
%OR 46.13  ; DONE ACQUIRE RFID NUMBER MANUAL
MOVL(498) &0 D500  ; NUMBER RFID DETECT
; rung 6
LD 45.13  ; REFRESH RFID HMI
OR P_First_Cycle
MOVL(498) #202D0000 D80  ; OUT HMI DISPLAY NO RFID
; rung 7
LD 13.12  ; START AUTO SEQUENCE
XFER(070) #2 D5000 D80  ; NUMBER RFID AUTO, OUT HMI DISPLAY NO RFID
; rung 8
LD 14.15  ; IR PH6
MOVL(498) #202D0000 D5000  ; NUMBER RFID AUTO
RSET 82.01  ; TURN ROT 1
RSET 82.02  ; TURN ROT 2
RSET 82.03  ; TURN ROT 3
RSET 82.04  ; TURN ROT 4
RSET 82.05  ; STRAIGHT ROT 4
; rung 9
LD 11.07  ; IR MANUAL
@AND 38.10  ; ENABLE RFID
MOVL(498) &0 D80  ; OUT HMI DISPLAY NO RFID

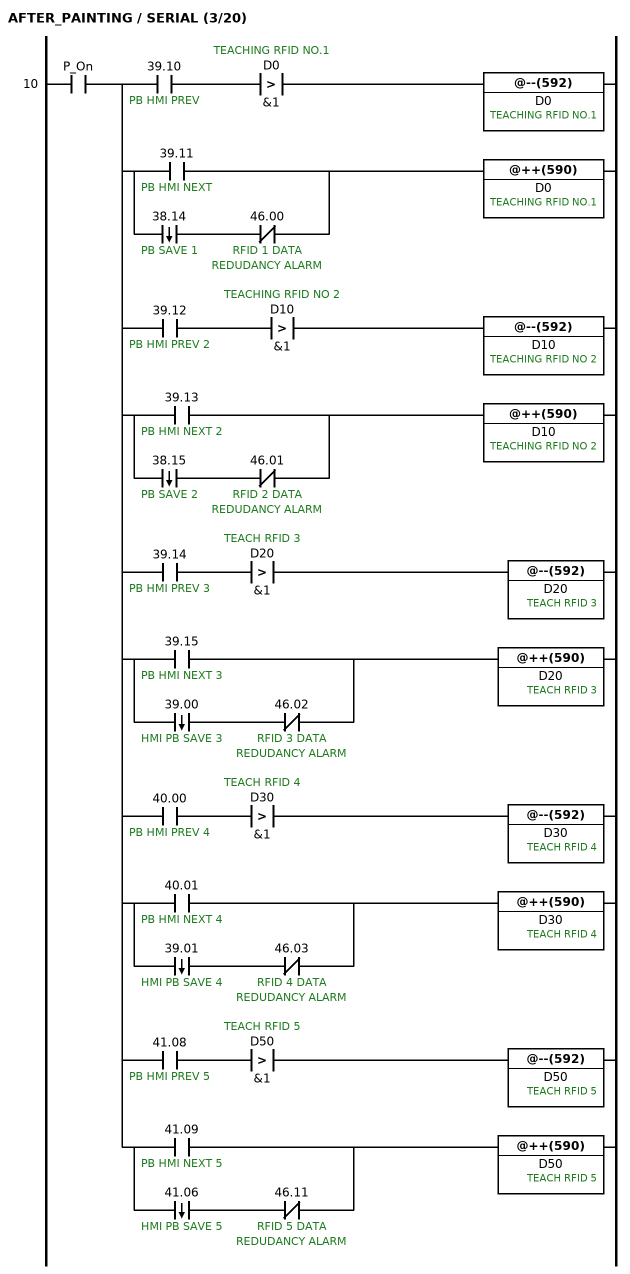
; rung 10
LD P_On
OUT TR0
AND 39.10  ; PB HMI PREV
AND>(320) D0 &1  ; TEACHING RFID NO.1
@--(592) D0  ; TEACHING RFID NO.1
LD TR0
LD 39.11  ; PB HMI NEXT
%LD 38.14  ; PB SAVE 1
ANDNOT 46.00  ; RFID 1 DATA REDUDANCY ALARM
ORLD
ANDLD
@++(590) D0  ; TEACHING RFID NO.1
LD TR0
AND 39.12  ; PB HMI PREV 2
AND>(320) D10 &1  ; TEACHING RFID NO 2
@--(592) D10  ; TEACHING RFID NO 2
LD TR0
LD 39.13  ; PB HMI NEXT 2
%LD 38.15  ; PB SAVE 2
ANDNOT 46.01  ; RFID 2 DATA REDUDANCY ALARM
ORLD
ANDLD
@++(590) D10  ; TEACHING RFID NO 2
LD TR0
AND 39.14  ; PB HMI PREV 3
AND>(320) D20 &1  ; TEACH RFID 3
@--(592) D20  ; TEACH RFID 3
LD TR0
LD 39.15  ; PB HMI NEXT 3
%LD 39.00  ; HMI PB SAVE 3
ANDNOT 46.02  ; RFID 3 DATA REDUDANCY ALARM
ORLD
ANDLD
@++(590) D20  ; TEACH RFID 3
LD TR0
AND 40.00  ; PB HMI PREV 4
AND>(320) D30 &1  ; TEACH RFID 4
@--(592) D30  ; TEACH RFID 4
LD TR0
LD 40.01  ; PB HMI NEXT 4
%LD 39.01  ; HMI PB SAVE 4
ANDNOT 46.03  ; RFID 4 DATA REDUDANCY ALARM
ORLD
ANDLD
@++(590) D30  ; TEACH RFID 4
LD TR0
AND 41.08  ; PB HMI PREV 5
AND>(320) D50 &1  ; TEACH RFID 5
@--(592) D50  ; TEACH RFID 5
LD TR0
LD 41.09  ; PB HMI NEXT 5
%LD 41.06  ; HMI PB SAVE 5
ANDNOT 46.11  ; RFID 5 DATA REDUDANCY ALARM
ORLD
ANDLD
@++(590) D50  ; TEACH RFID 5

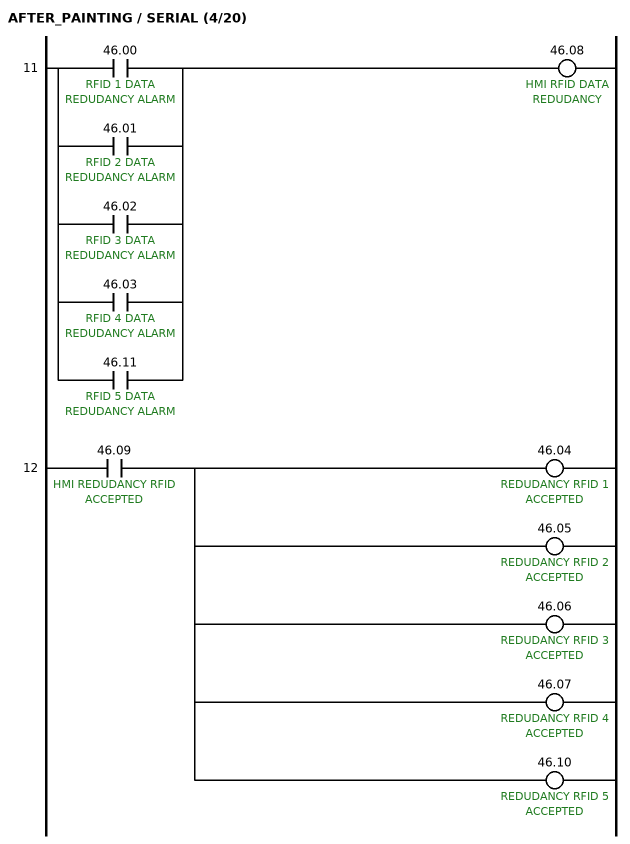
; rung 11
LD 46.00  ; RFID 1 DATA REDUDANCY ALARM
OR 46.01  ; RFID 2 DATA REDUDANCY ALARM
OR 46.02  ; RFID 3 DATA REDUDANCY ALARM
OR 46.03  ; RFID 4 DATA REDUDANCY ALARM
OR 46.11  ; RFID 5 DATA REDUDANCY ALARM
OUT 46.08  ; HMI RFID DATA REDUDANCY
; rung 12
LD 46.09  ; HMI REDUDANCY RFID ACCEPTED
OUT 46.04  ; REDUDANCY RFID 1 ACCEPTED
OUT 46.05  ; REDUDANCY RFID 2 ACCEPTED
OUT 46.06  ; REDUDANCY RFID 3 ACCEPTED
OUT 46.07  ; REDUDANCY RFID 4 ACCEPTED
OUT 46.10  ; REDUDANCY RFID 5 ACCEPTED

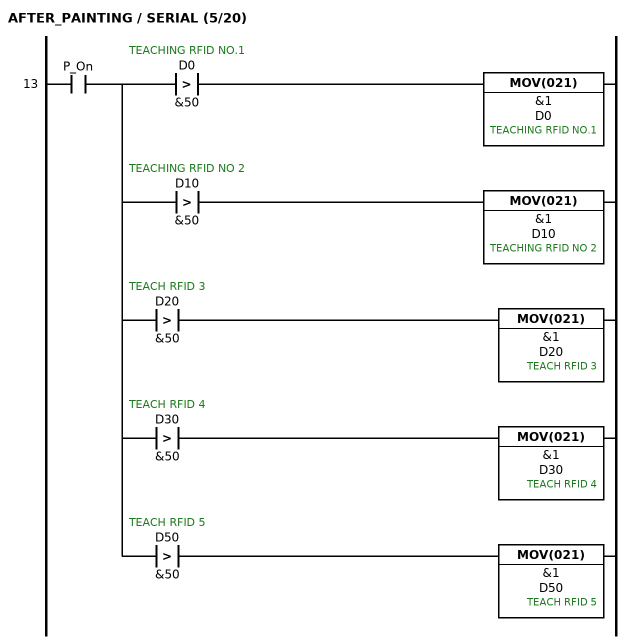
; rung 13
LD P_On
OUT TR0
AND>(320) D0 &50  ; TEACHING RFID NO.1
MOV(021) &1 D0  ; TEACHING RFID NO.1
LD TR0
AND>(320) D10 &50  ; TEACHING RFID NO 2
MOV(021) &1 D10  ; TEACHING RFID NO 2
LD TR0
AND>(320) D20 &50  ; TEACH RFID 3
MOV(021) &1 D20  ; TEACH RFID 3
LD TR0
AND>(320) D30 &50  ; TEACH RFID 4
MOV(021) &1 D30  ; TEACH RFID 4
LD TR0
AND>(320) D50 &50  ; TEACH RFID 5
MOV(021) &1 D50  ; TEACH RFID 5

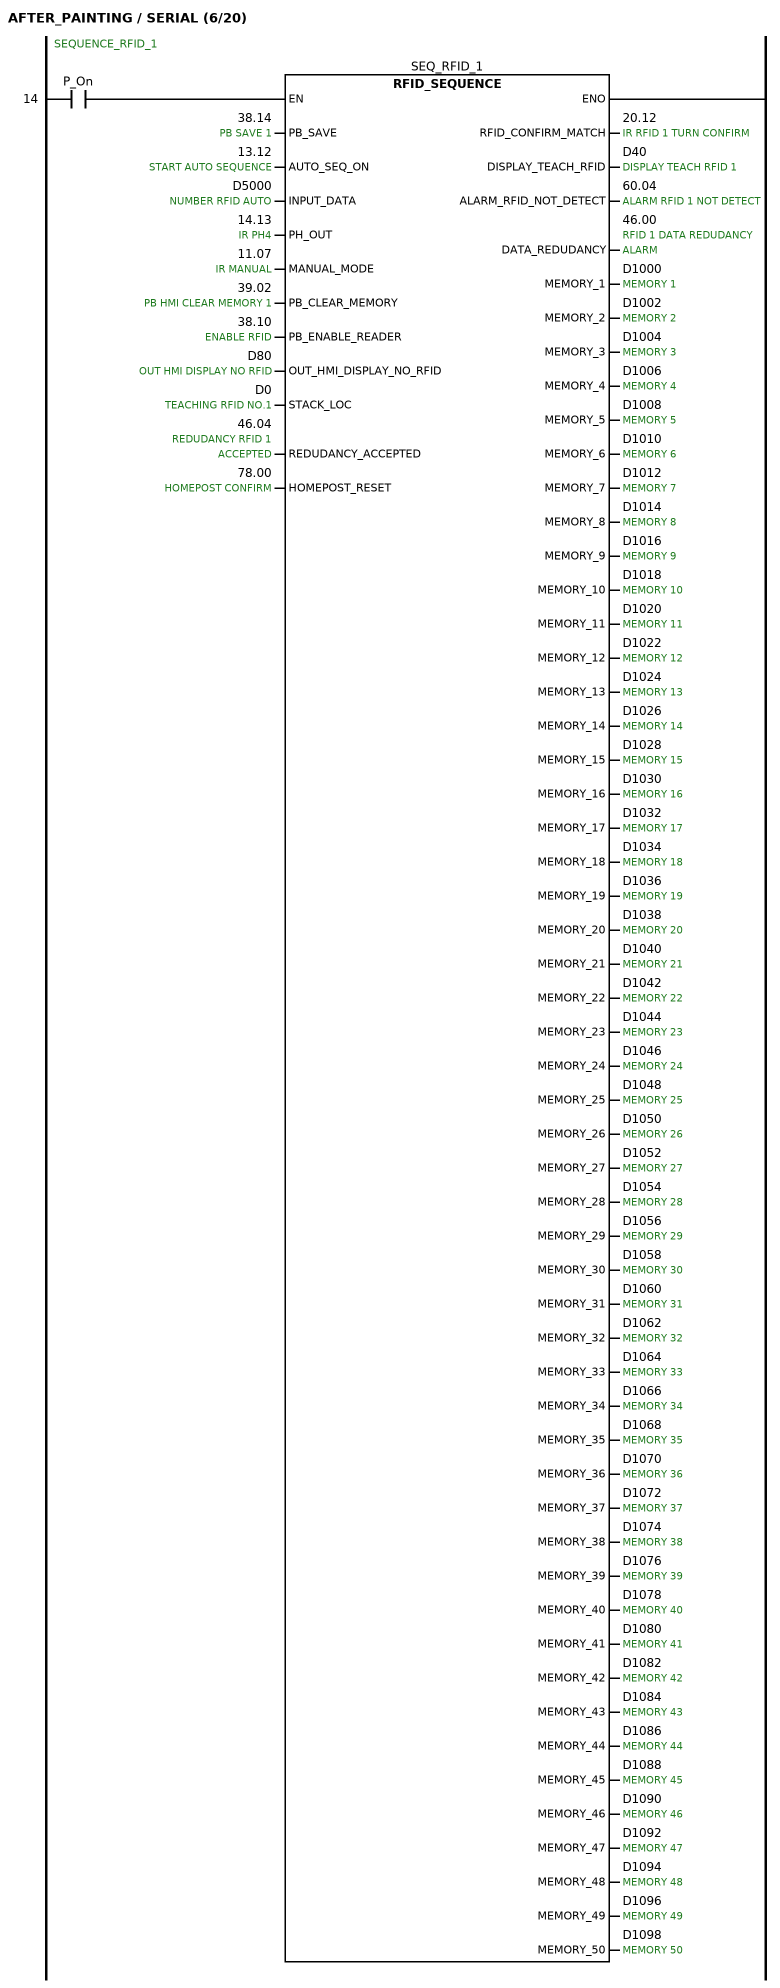
; rung 14: SEQUENCE_RFID_1
LD P_On
CALL SEQ_RFID_1 : RFID_SEQUENCE (PB_SAVE := 38.14, AUTO_SEQ_ON := 13.12, INPUT_DATA := D5000, PH_OUT := 14.13, MANUAL_MODE := 11.07, PB_CLEAR_MEMORY := 39.02, PB_ENABLE_READER := 38.10, OUT_HMI_DISPLAY_NO_RFID := D80, STACK_LOC := D0, REDUDANCY_ACCEPTED := 46.04, HOMEPOST_RESET := 78.00, RFID_CONFIRM_MATCH => 20.12, DISPLAY_TEACH_RFID => D40, ALARM_RFID_NOT_DETECT => 60.04, DATA_REDUDANCY => 46.00, MEMORY_1 => D1000, MEMORY_2 => D1002, MEMORY_3 => D1004, MEMORY_4 => D1006, MEMORY_5 => D1008, MEMORY_6 => D1010, MEMORY_7 => D1012, MEMORY_8 => D1014, MEMORY_9 => D1016, MEMORY_10 => D1018, MEMORY_11 => D1020, MEMORY_12 => D1022, MEMORY_13 => D1024, MEMORY_14 => D1026, MEMORY_15 => D1028, MEMORY_16 => D1030, MEMORY_17 => D1032, MEMORY_18 => D1034, MEMORY_19 => D1036, MEMORY_20 => D1038, MEMORY_21 => D1040, MEMORY_22 => D1042, MEMORY_23 => D1044, MEMORY_24 => D1046, MEMORY_25 => D1048, MEMORY_26 => D1050, MEMORY_27 => D1052, MEMORY_28 => D1054, MEMORY_29 => D1056, MEMORY_30 => D1058, MEMORY_31 => D1060, MEMORY_32 => D1062, MEMORY_33 => D1064, MEMORY_34 => D1066, MEMORY_35 => D1068, MEMORY_36 => D1070, MEMORY_37 => D1072, MEMORY_38 => D1074, MEMORY_39 => D1076, MEMORY_40 => D1078, MEMORY_41 => D1080, MEMORY_42 => D1082, MEMORY_43 => D1084, MEMORY_44 => D1086, MEMORY_45 => D1088, MEMORY_46 => D1090, MEMORY_47 => D1092, MEMORY_48 => D1094, MEMORY_49 => D1096, MEMORY_50 => D1098)  ; PB SAVE 1, START AUTO SEQUENCE, NUMBER RFID AUTO, IR PH4, IR MANUAL, PB HMI CLEAR MEMORY 1, ENABLE RFID, OUT HMI DISPLAY NO RFID, TEACHING RFID NO.1, REDUDANCY RFID 1 ACCEPTED, HOMEPOST CONFIRM, IR RFID 1 TURN CONFIRM, DISPLAY TEACH RFID 1, ALARM RFID 1 NOT DETECT, RFID 1 DATA REDUDANCY ALARM, MEMORY 1, MEMORY 2, MEMORY 3, MEMORY 4, MEMORY 5, MEMORY 6, MEMORY 7, MEMORY 8, MEMORY 9, MEMORY 10, MEMORY 11, MEMORY 12, MEMORY 13, MEMORY 14, MEMORY 15, MEMORY 16, MEMORY 17, MEMORY 18, MEMORY 19, MEMORY 20, MEMORY 21, MEMORY 22, MEMORY 23, MEMORY 24, MEMORY 25, MEMORY 26, MEMORY 27, MEMORY 28, MEMORY 29, MEMORY 30, MEMORY 31, MEMORY 32, MEMORY 33, MEMORY 34, MEMORY 35, MEMORY 36, MEMORY 37, MEMORY 38, MEMORY 39, MEMORY 40, MEMORY 41, MEMORY 42, MEMORY 43, MEMORY 44, MEMORY 45, MEMORY 46, MEMORY 47, MEMORY 48, MEMORY 49, MEMORY 50

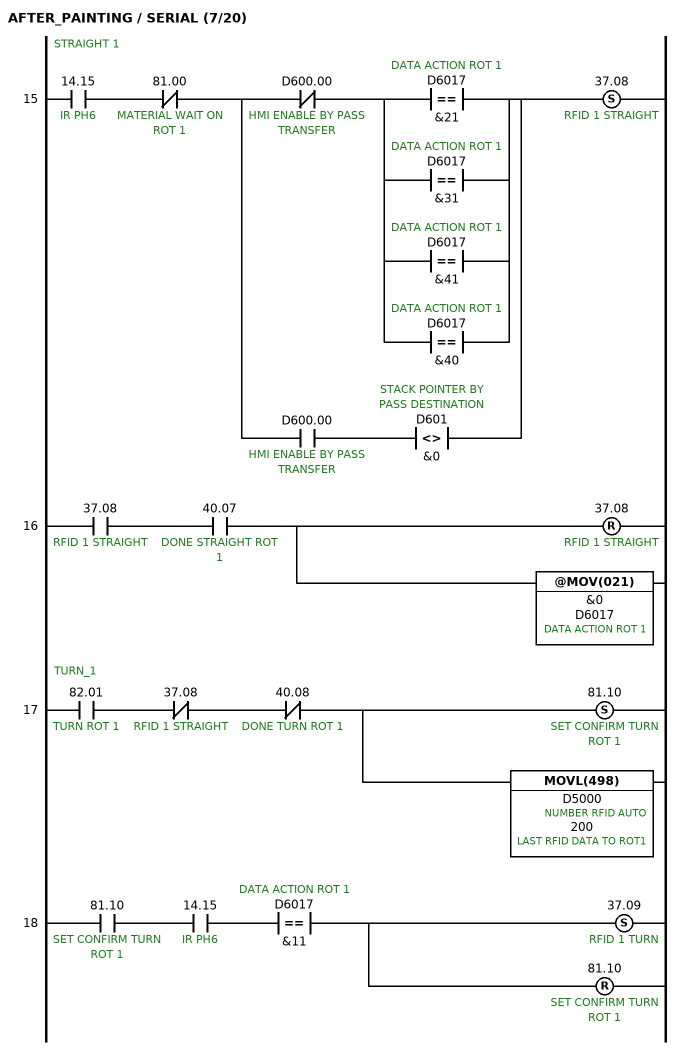
; rung 15: STRAIGHT 1
LD 14.15  ; IR PH6
ANDNOT 81.00  ; MATERIAL WAIT ON ROT 1
LDNOT D600.00  ; HMI ENABLE BY PASS TRANSFER
LD=(300) D6017 &21  ; DATA ACTION ROT 1
OR=(300) D6017 &31  ; DATA ACTION ROT 1
OR=(300) D6017 &41  ; DATA ACTION ROT 1
OR=(300) D6017 &40  ; DATA ACTION ROT 1
ANDLD
LD D600.00  ; HMI ENABLE BY PASS TRANSFER
AND<>(305) D601 &0  ; STACK POINTER BY PASS DESTINATION
ORLD
ANDLD
SET 37.08  ; RFID 1 STRAIGHT
; rung 16
LD 37.08  ; RFID 1 STRAIGHT
AND 40.07  ; DONE STRAIGHT ROT 1
RSET 37.08  ; RFID 1 STRAIGHT
@MOV(021) &0 D6017  ; DATA ACTION ROT 1
; rung 17: TURN_1
LD 82.01  ; TURN ROT 1
ANDNOT 37.08  ; RFID 1 STRAIGHT
ANDNOT 40.08  ; DONE TURN ROT 1
SET 81.10  ; SET CONFIRM TURN ROT 1
MOVL(498) D5000 200  ; NUMBER RFID AUTO, LAST RFID DATA TO ROT1
; rung 18
LD 81.10  ; SET CONFIRM TURN ROT 1
AND 14.15  ; IR PH6
AND=(300) D6017 &11  ; DATA ACTION ROT 1
SET 37.09  ; RFID 1 TURN
RSET 81.10  ; SET CONFIRM TURN ROT 1

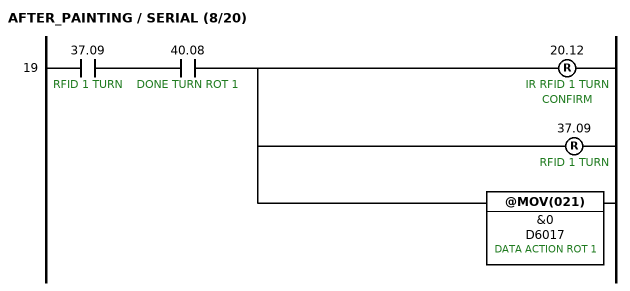
; rung 19
LD 37.09  ; RFID 1 TURN
AND 40.08  ; DONE TURN ROT 1
RSET 20.12  ; IR RFID 1 TURN CONFIRM
RSET 37.09  ; RFID 1 TURN
@MOV(021) &0 D6017  ; DATA ACTION ROT 1

